(* IEC 61131-3 sources: plc_generation_empirical_study/datasets/task_bank_c04_reverse_runtime_v0_3/tasks/C04_S16_lean_composite, 2 files *)

(* ---- interface.st ---- *)
FUNCTION_BLOCK C04_S16_lean_composite
VAR_INPUT
    A_AutoMode : BOOL;
    A_AutoDemand : BOOL;
    A_ManualDemand : BOOL;
    A_SafetyOK : BOOL;
    A_Inhibit : BOOL;
    B_Event : BOOL;
    B_Qualify : BOOL;
    B_Reset : BOOL;
    B_MaxCount : INT;
    SubsystemBEnable : BOOL;
    CrossReset : BOOL;
END_VAR
VAR_OUTPUT
    A_Command : BOOL;
    A_Blocked : BOOL;
    B_Count : INT;
    B_AcceptedPulse : BOOL;
    B_AtLimit : BOOL;
    CrossReady : BOOL;
    CrossBlocked : BOOL;
END_VAR
END_FUNCTION_BLOCK

(* ---- reference.st ---- *)
FUNCTION_BLOCK C04_S16_lean_composite
VAR_INPUT
    A_AutoMode : BOOL;
    A_AutoDemand : BOOL;
    A_ManualDemand : BOOL;
    A_SafetyOK : BOOL;
    A_Inhibit : BOOL;
    B_Event : BOOL;
    B_Qualify : BOOL;
    B_Reset : BOOL;
    B_MaxCount : INT;
    SubsystemBEnable : BOOL;
    CrossReset : BOOL;
END_VAR
VAR_OUTPUT
    A_Command : BOOL;
    A_Blocked : BOOL;
    B_Count : INT;
    B_AcceptedPulse : BOOL;
    B_AtLimit : BOOL;
    CrossReady : BOOL;
    CrossBlocked : BOOL;
END_VAR
VAR
    B_PrevEvent : BOOL := FALSE;
END_VAR

A_Command := ((A_AutoMode AND A_AutoDemand) OR ((NOT A_AutoMode) AND A_ManualDemand))
           AND A_SafetyOK AND (NOT A_Inhibit);
A_Blocked := ((A_AutoMode AND A_AutoDemand) OR ((NOT A_AutoMode) AND A_ManualDemand))
           AND ((NOT A_SafetyOK) OR A_Inhibit);

IF CrossReset THEN
    CrossReady := FALSE;
ELSIF A_Command THEN
    CrossReady := TRUE;
END_IF;
CrossBlocked := SubsystemBEnable AND (NOT CrossReady);

IF SubsystemBEnable AND CrossReady THEN
    B_AcceptedPulse := FALSE;
    IF B_Reset THEN
        B_Count := 0;
    ELSIF B_Event AND (NOT B_PrevEvent) AND B_Qualify AND (B_Count < B_MaxCount) THEN
        B_Count := B_Count + 1;
        B_AcceptedPulse := TRUE;
    END_IF;
    B_AtLimit := B_Count >= B_MaxCount;
    B_PrevEvent := B_Event;
ELSE
    B_Count := 0;
    B_AcceptedPulse := FALSE;
    B_AtLimit := FALSE;
END_IF;

END_FUNCTION_BLOCK
